// TwinCAT 3 PLC project Untitled1
// ProgramVersion: 3.1.4022.4
// libraries:
//   Tc2_Standard, * (Beckhoff Automation GmbH)
//   Tc2_System, * (Beckhoff Automation GmbH)
//   Tc3_Module, * (Beckhoff Automation GmbH)
// project tree:
//   / PlcTask.TcTTO
//   POUs/ MAIN.TcPOU

CONFIGURATION Untitled1
    RESOURCE PLC ON TwinCAT3
        TASK PlcTask(INTERVAL := T#10ms, PRIORITY := 20);
        PROGRAM MAIN WITH PlcTask : MAIN;
    END_RESOURCE
END_CONFIGURATION

// ---- POUs/MAIN.TcPOU
PROGRAM MAIN
VAR
	{attribute 'OPC.UA.DA' := '1'}
	SensoreStart AT %M* : BOOL := FALSE;
	{attribute 'OPC.UA.DA' := '1'}
	SensoreReset AT %M* : BOOL := FALSE;
	{attribute 'OPC.UA.DA' := '1'}
	SensoreFCD0 AT %M* : BOOL := FALSE;
	{attribute 'OPC.UA.DA' := '1'}
	SensoreFCD1P AT %M* : BOOL := FALSE;
	{attribute 'OPC.UA.DA' := '1'}
	SensoreFCDPP AT %M* : BOOL := FALSE;
	{attribute 'OPC.UA.DA' := '1'}
	SensoreFCD2P AT %M* : BOOL := FALSE;
	{attribute 'OPC.UA.DA' := '1'}
	SensoreFCD3P AT %M* : BOOL := FALSE;
	{attribute 'OPC.UA.DA' := '1'}
	SensoreFCDCP AT %M* : BOOL := FALSE;
	{attribute 'OPC.UA.DA' := '1'}
	SensoreFCD1V AT %M* : BOOL := FALSE;
	{attribute 'OPC.UA.DA' := '1'}
	SensoreFCDPV AT %M* : BOOL := FALSE;
	{attribute 'OPC.UA.DA' := '1'}
	SensoreFCD2V AT %M* : BOOL := FALSE;
	{attribute 'OPC.UA.DA' := '1'}
	SensoreFCD3V AT %M* : BOOL := FALSE;
	{attribute 'OPC.UA.DA' := '1'}
	SensoreFCDCV AT %M* : BOOL := FALSE;
	{attribute 'OPC.UA.DA' := '1'}
	Random AT %M* : BOOL;
	{attribute 'OPC.UA.DA' := '1'}
	PP AT %M* : BOOL := FALSE;
	{attribute 'OPC.UA.DA' := '1'}
	PV AT %M* : BOOL := FALSE;
	{attribute 'OPC.UA.DA' := '1'}
	ComandoDX AT %M* : BOOL := FALSE;
	{attribute 'OPC.UA.DA' := '1'}
	ComandoDX2P AT %M* : BOOL := FALSE;
	{attribute 'OPC.UA.DA' := '1'}
	ComandoDX2V AT %M* : BOOL := FALSE;
	{attribute 'OPC.UA.DA' := '1'}
	ComandoDX3P AT %M* : BOOL := FALSE;
	{attribute 'OPC.UA.DA' := '1'}
	ComandoDX3V AT %M* : BOOL := FALSE;
	{attribute 'OPC.UA.DA' := '1'}
	ComandoPressaP AT %M* : BOOL := FALSE;
	{attribute 'OPC.UA.DA' := '1'}
    ComandoPressaV AT %M* : BOOL := FALSE;
	{attribute 'OPC.UA.DA' := '1'}
	ComandoCamionP AT %M* : BOOL := FALSE;
	{attribute 'OPC.UA.DA' := '1'}
	ComandoCamionV AT %M* : BOOL := FALSE;
	{attribute 'OPC.UA.DA' := '1'}
	ComandoAlarm AT %M* : BOOL := FALSE;
	{attribute 'OPC.UA.DA' := '1'}
	TimeWatchDog AT %M* : TIME := T#10S;
	{attribute 'OPC.UA.DA' := '1'}
	TimeAct AT %M* : TIME := T#0S;
	{attribute 'OPC.UA.DA' := '1'}
	TimeAct2 AT %M* : TIME := T#0S;
	
	fbTIMER AT %M* : TON;
	fbTIMER2 AT %M* : TON;

END_VAR

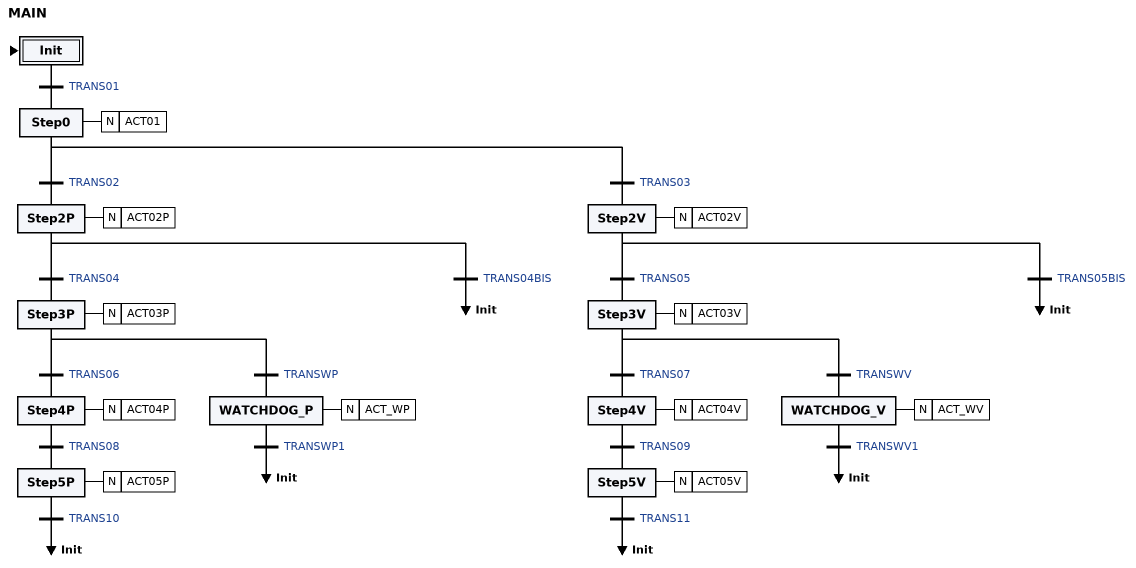
INITIAL_STEP Init:
END_STEP
TRANSITION FROM Init TO Step0
    := TRANS01;
END_TRANSITION
STEP Step0:
    ACT01(N);
END_STEP
TRANSITION FROM Step0 TO Step2P
    := TRANS02;
END_TRANSITION
STEP Step2P:
    ACT02P(N);
END_STEP
TRANSITION FROM Step2P TO Step3P
    := TRANS04;
END_TRANSITION
TRANSITION FROM Step2P TO Init
    := TRANS04BIS;
END_TRANSITION
STEP Step3P:
    ACT03P(N);
END_STEP
TRANSITION FROM Step3P TO Step4P
    := TRANS06;
END_TRANSITION
TRANSITION FROM Step3P TO WATCHDOG_P
    := TRANSWP;
END_TRANSITION
STEP WATCHDOG_P:
    ACT_WP(N);
END_STEP
TRANSITION FROM WATCHDOG_P TO Init
    := TRANSWP1;
END_TRANSITION
STEP Step4P:
    ACT04P(N);
END_STEP
TRANSITION FROM Step4P TO Step5P
    := TRANS08;
END_TRANSITION
STEP Step5P:
    ACT05P(N);
END_STEP
TRANSITION FROM Step5P TO Init
    := TRANS10;
END_TRANSITION
TRANSITION FROM Step0 TO Step2V
    := TRANS03;
END_TRANSITION
STEP Step2V:
    ACT02V(N);
END_STEP
TRANSITION FROM Step2V TO Step3V
    := TRANS05;
END_TRANSITION
TRANSITION FROM Step2V TO Init
    := TRANS05BIS;
END_TRANSITION
STEP Step3V:
    ACT03V(N);
END_STEP
TRANSITION FROM Step3V TO Step4V
    := TRANS07;
END_TRANSITION
TRANSITION FROM Step3V TO WATCHDOG_V
    := TRANSWV;
END_TRANSITION
STEP WATCHDOG_V:
    ACT_WV(N);
END_STEP
TRANSITION FROM WATCHDOG_V TO Init
    := TRANSWV1;
END_TRANSITION
STEP Step4V:
    ACT04V(N);
END_STEP
TRANSITION FROM Step4V TO Step5V
    := TRANS09;
END_TRANSITION
STEP Step5V:
    ACT05V(N);
END_STEP
TRANSITION FROM Step5V TO Init
    := TRANS11;
END_TRANSITION

ACTION ACT_WP:
ComandoAlarm := TRUE;
END_ACTION

ACTION ACT_WV:
ComandoAlarm := TRUE;
END_ACTION

ACTION ACT01:
ComandoDX := TRUE; 

ComandoAlarm := FALSE;
ComandoDX2P := FALSE; 
ComandoDX2V := FALSE; 
ComandoCamionP :=FALSE;
ComandoCamionV :=FALSE;

ComandoPressaP := FALSE;
ComandoPressaV := FALSE;

fbTIMER2(IN:= FALSE , PT:= TimeWatchDog);
TimeAct2 := fbTIMER2.ET;

fbTIMER(IN:= FALSE , PT:= TimeWatchDog);
TimeAct := fbTIMER.ET;
END_ACTION

ACTION ACT02P:
ComandoDX2P := TRUE;
ComandoDX := FALSE;
END_ACTION

ACTION ACT02V:
ComandoDX2V := TRUE;
ComandoDX := FALSE;
END_ACTION

ACTION ACT03P:
ComandoPressaP:= TRUE;

ComandoDX2P := FALSE;
fbTIMER(IN:= TRUE , PT:= TimeWatchDog);
TimeAct := fbTIMER.ET;
END_ACTION

ACTION ACT03V:
ComandoPressaV:= TRUE;

ComandoDX2V := FALSE;
fbTIMER2(IN:= TRUE , PT:= TimeWatchDog);
TimeAct2 := fbTIMER2.ET;
END_ACTION

ACTION ACT04P:
ComandoDX3P := TRUE;
ComandoPressaP := FALSE;
END_ACTION

ACTION ACT04V:
ComandoDX3V := TRUE;
ComandoPressaV := FALSE;
END_ACTION

ACTION ACT05P:
ComandoCamionP := TRUE;
ComandoDX3P := FALSE;
END_ACTION

ACTION ACT05V:
ComandoCamionV := TRUE;
ComandoDX3V := FALSE;
END_ACTION

TRANSITION TRANS01:
SensoreStart;
END_TRANSITION

TRANSITION TRANS02:
SensoreFCD1P;
END_TRANSITION

TRANSITION TRANS03:
SensoreFCD1V;
END_TRANSITION

TRANSITION TRANS04:
SensoreFCDPP;
END_TRANSITION

TRANSITION TRANS04BIS:
PP;
END_TRANSITION

TRANSITION TRANS05:
SensoreFCDPV;
END_TRANSITION

TRANSITION TRANS05BIS:
PV;
END_TRANSITION

TRANSITION TRANS06:
SensoreFCD2P;
END_TRANSITION

TRANSITION TRANS07:
SensoreFCD2V;
END_TRANSITION

TRANSITION TRANS08:
SensoreFCD3P;
END_TRANSITION

TRANSITION TRANS09:
SensoreFCD3V;
END_TRANSITION

TRANSITION TRANS10:
SensoreFCDCP;
END_TRANSITION

TRANSITION TRANS11:
SensoreFCDCV;
END_TRANSITION

TRANSITION TRANSWP:
fbTIMER.Q;
END_TRANSITION

TRANSITION TRANSWP1:
SensoreReset;
END_TRANSITION

TRANSITION TRANSWV:
fbTIMER2.Q ;
END_TRANSITION

TRANSITION TRANSWV1:
SensoreReset;
END_TRANSITION

END_PROGRAM
